FUNCTION_BLOCK ValveControlSR (* Basic Function Block Type *)
  (* Standard: 61499-2 *)
  (* Version 0.0, 5/28/2016, Andrei, nxtControl GmbH, Template *)
  PACKAGE Main;
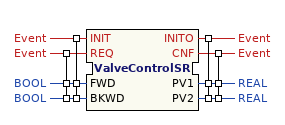
  EVENT_INPUT
    INIT WITH FWD, BKWD; (* Initialization Request *)
    REQ WITH FWD, BKWD; (* Normal Execution Request *)
  END_EVENT
  EVENT_OUTPUT
    INITO WITH PV1, PV2; (* Initialization Confirm *)
    CNF WITH PV1, PV2; (* Execution Confirmation *)
  END_EVENT
  VAR_INPUT
    FWD : BOOL; (* Input event qualifier *)
    BKWD : BOOL;
  END_VAR
  VAR_OUTPUT
    PV1 : REAL; (* Output event qualifier *)
    PV2 : REAL;
  END_VAR
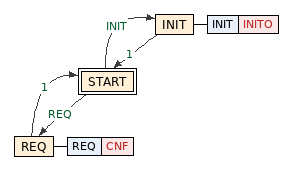
  EC_STATES
    START; (* Initial State *)
    INIT : INIT -> INITO; (* Initialization *)
    REQ : REQ -> CNF; (* Normal execution *)
  END_STATES
  EC_TRANSITIONS
    START TO INIT := INIT;
    INIT TO START := 1;
    START TO REQ := REQ;
    REQ TO START := 1;
  END_TRANSITIONS
  ALGORITHM INIT IN ST: (* Initialization algorithm *)
PV1 := 0.0;
PV2 := 0.0;
  END_ALGORITHM
  ALGORITHM REQ IN ST: (* Normally executed algorithm *)
IF FWD AND NOT(BKWD) THEN
	PV1 := 200;
	PV2 := 0.0;
ELSIF NOT(FWD) AND BKWD THEN
	PV1 := 0.0;
	PV2 := 200.0;
ELSE
	PV1 := 0.0;
	PV2 := 0.0;
END_IF;
  END_ALGORITHM
END_FUNCTION_BLOCK
